// TIA Portal V18 export
DATA_BLOCK "TON"   // DB163
{ S7_Optimized_Access := 'TRUE' }
VERSION : 0.1
// stored: AutoNumber false, DBAccessibleFromOPCUA true, DBAccessibleFromWebserver true, IsOnlyStoredInLoadMemory false, IsRetainMemResEnabled false, IsWriteProtectedInAS false, MemoryReserve 100
   VAR
      TON : Array[0..100] of TON_TIME;
      CTU { S7_SetPoint := 'True'} : Array[0..20] of IEC_DCOUNTER;
   END_VAR
   VAR RETAIN
      P { S7_SetPoint := 'True'} : Array[0..20] of Bool;
   END_VAR
BEGIN
END_DATA_BLOCK
